// TIA Portal V21 export
TYPE "Std_Comunicazione"
   STRUCT
      Prm : Struct
         PutEnabled : Bool;
         GetEnabled : Bool;
         "Timer" : Struct
            PutTimeOut : "Std_stTimer";
            PutExecuteDelay { S7_SetPoint := 'True'} : "Std_stTimer";
            GetTimeOut { S7_SetPoint := 'True'} : "Std_stTimer";
            GetExecuteDelay { S7_SetPoint := 'True'} : "Std_stTimer";
         END_STRUCT;
      END_STRUCT;
      Hmi : Struct
         Diagnostica : Struct
            "0-" : Bool;
            "1-" : Bool;
            "2-" : Bool;
            "3-" : Bool;
            "4-" : Bool;
            "5-" : Bool;
            "6-" : Bool;
            "7-" : Bool;
            "8-" : Bool;
            "9-" : Bool;
         END_STRUCT;
      END_STRUCT;
      Dati { S7_SetPoint := 'True'} : "Std_DatiGetPut";
      Allarmi : Struct
         TimeOutCom : "Std_stTimer";
         Stato : Struct
            PUT_Alarm : Bool;
            Get_Alarm : Bool;
            PUT_AlarmCode : Word;
            Get_AlarmCode : Word;
            Watchdog : Bool;
         END_STRUCT;
         EnCadutaCiclo : Struct   // Abilita la caduta del ciclo di riferimento per allarme corrispondente
            PUT_Alarm : Bool;
            Get_Alarm : Bool;
            Watchdog : Bool;
         END_STRUCT;
         WordHMI : Word;   // Word per lista segnalazioni HMI
      END_STRUCT;
   END_STRUCT;
END_TYPE
